Staubli VAL3: ros_server.pjx

--- ros_server.pjx ---
Parameters version=s7.7.2 stackSize=5000 millimeterUnit=true
Program file=atan2.pgx
Program file=dataReceiver.pgx
Program file=dataStreamer.pgx
Program file=decodeMsgBody.pgx
Program file=decodeMsgHeader.pgx
Program file=decTrajPtCartesian.pgx
Program file=decTrajPtJoint.pgx
Program file=decTrajPtJointFull.pgx
Program file=encodeAck.pgx
Program file=encodeJState.pgx
Program file=encodeStatus.pgx
Program file=encPrefixHeader.pgx
Program file=encTrajPtCartesianAck.pgx
Program file=encTrajPtJointAck.pgx
Program file=encTrajPtJointFAck.pgx
Program file=fetchStatus.pgx
Program file=initParams.pgx
Program file=motionControl.pgx
Program file=pushMotion.pgx
Program file=recvData.pgx
Program file=recvHeartbeat.pgx
Program file=recvMsgBody.pgx
Program file=recvMsgHeader.pgx
Program file=recvTrajPtCartesian.pgx
Program file=recvTrajPtJoint.pgx
Program file=recvTrajPtJointFull.pgx
Program file=screenUpdate.pgx
Program file=sendAck.pgx
Program file=sendData.pgx
Program file=sendRosMsg.pgx
Program file=setupRosMsgs.pgx
Program file=start.pgx
Program file=stop.pgx
Program file=toJointArrayRad.pgx
Program file=toJointRxDeg.pgx
Program file=toPointRxEuler.pgx
Program file=toPointRxMillis.pgx
Data file=ros_server.dtx
Library alias=libQueueFuncs path=Disk://ros_libs/QueueFuncs/QueueFuncs.pjx
Type name=RosSimpleMsg path=Disk://ros_libs/RosSimpleMsg/RosSimpleMsg.pjx
Type name=RobotStatusMsg path=Disk://ros_libs/RobotStatusMsg/RobotStatusMsg.pjx
Type name=CartesianTrajPtMsg path=Disk://ros_libs/CartesianTrajPtMsg/CartesianTrajPtMsg.pjx
Type name=JointStateMsg path=Disk://ros_libs/JointStateMsg/JointStateMsg.pjx
Type name=JointTrajPtMsg path=Disk://ros_libs/JointTrajPtMsg/JointTrajPtMsg.pjx
Type name=JointTrajPtFMsg path=Disk://ros_libs/JointTrajPtFMsg/JointTrajPtFMsg.pjx
Type name=JointFbkMsg path=Disk://ros_libs/JointFbkMsg/JointFbkMsg.pjx
Type name=MotionCmd path=Disk://ros_libs/MotionCmd/MotionCmd.pjx
Type name=Header path=Disk://ros_libs/Header/Header.pjx
Type name=Prefix path=Disk://ros_libs/Prefix/Prefix.pjx
Type name=Body path=Disk://ros_libs/Body/Body.pjx
Type name=Queue path=Disk://ros_libs/Queue/Queue.pjx

--- ros_server.dtx ---
public bool bFbkOverrun
public bool bMotionOverrun
public sio siTcpIpFbk = {link=Socket\Feedback}
public sio siTcpIpMotion = {link=Socket\Motion}
public string sStreamTaskName = "publisher"
public string sMotionTaskName
public RosSimpleMsg rosGenericMsg
  [0]
    Header header
      [0]
        num nMsgType
        num nCommType
        num nReplyCode
        num nData[12]
    Prefix prefix
      [0]
        num nLength
        num nData[4]
public tool tTool = {fatherId=flange[0], ioLink=valve1}
public string sTrajPtTaskName
public bool bTrajPtOverrun
public RobotStatusMsg rosStatusMsg
  [0]
    Body body
      [0]
        num nData[28]
    Header header
      [0]
        num nMsgType
        num nCommType
        num nReplyCode
        num nData[12]
    Prefix prefix
      [0]
        num nLength
        num nData[4]
    RobotStatus robotStatus
      [0]
        num nDrivesPowered
        num nEStopped
        num nErrorCode
        num nInError
        num nInMotion
        num nMode
        num nMotionPossible
public JointStateMsg rosJointMsg
  [0]
    Header header
      [0]
        num nMsgType
        num nCommType
        num nReplyCode
        num nData[12]
    Body body
      [0]
        num nData[44]
    JointState jointState
      [0]
        num nSeq
        num nJoints[10]
    Prefix prefix
      [0]
        num nLength
        num nData[4]
public JointTrajPtMsg rosTrajPtMsg
  [0]
    Header header
      [0]
        num nMsgType
        num nCommType
        num nReplyCode
        num nData[12]
    JointTrajPt jointTrajPt
      [0]
        num nSeq
        num nJoints[10]
        num nVelocity
        num nDuration
    Prefix prefix
      [0]
        num nLength
        num nData[4]
    Body body
      [0]
        num nData[52]
public JointTrajPtFMsg rosTrajPtFMsg
  [0]
    Header header
      [0]
        num nMsgType
        num nCommType
        num nReplyCode
        num nData[12]
    Prefix prefix
      [0]
        num nLength
        num nData[4]
    JointTrajPtFull jointTrajPtFull
      [0]
        num nRobotId
        num nSeq
        num nValidFields
        num nTime
        num nPositions[10]
        num nVelocities[10]
        num nAccelerations[10]
    Body body
      [0]
        num nData[136]
public JointFbkMsg rosJointFbkMsg
  [0]
    Header header
      [0]
        num nMsgType
        num nCommType
        num nReplyCode
        num nData[12]
    Prefix prefix
      [0]
        num nLength
        num nData[4]
    JointFeedback jointFeedback
      [0]
        num nRobotId
        num nValidFields
        num nTime
        num nPositions[10]
        num nVelocities[10]
        num nAccelerations[10]
    Body body
      [0]
        num nData[132]
public JointTrajPtFMsg rosTrajPtFAck
  [0]
    Header header
      [0]
        num nMsgType
        num nCommType
        num nReplyCode
        num nData[12]
    Prefix prefix
      [0]
        num nLength
        num nData[4]
    JointTrajPtFull jointTrajPtFull
      [0]
        num nRobotId
        num nSeq
        num nValidFields
        num nTime
        num nPositions[10]
        num nVelocities[10]
        num nAccelerations[10]
    Body body
      [0]
        num nData[136]
public JointTrajPtMsg rosTrajPtAck
  [0]
    Header header
      [0]
        num nMsgType
        num nCommType
        num nReplyCode
        num nData[12]
    JointTrajPt jointTrajPt
      [0]
        num nSeq
        num nJoints[10]
        num nVelocity
        num nDuration
    Prefix prefix
      [0]
        num nLength
        num nData[4]
    Body body
      [0]
        num nData[52]
public bool bScreenOverrun
public string sScreenTaskName
public num nInConnFlag
public num nOutConnFlag
public screen scDebug
public screen scMonitor
public string sHtbtTaskName
public num nPtsPopped
public bool bStopNow
public num nMotionProgress
public num nMoveId
public num nMovePts
public num nElapsedTime
public num nHeaderTime
public bool bOverwriteVel
public Queue qMoveBuffer
  [0]
    num nPush
    num nPop
    num nElems
    MotionCmd buffer[10]
      [0]
        mdesc mDesc = {leave=0, reach=0}
        num nDuration
        num nSequence
        num nMoveType
        jointRx jJointRx
        pointRx pPointRx
      [1]
        mdesc mDesc = {leave=0, reach=0}
        num nDuration
        num nSequence
        num nMoveType
        jointRx jJointRx
        pointRx pPointRx
      [2]
        mdesc mDesc = {leave=0, reach=0}
        num nDuration
        num nSequence
        num nMoveType
        jointRx jJointRx
        pointRx pPointRx
      [3]
        mdesc mDesc = {leave=0, reach=0}
        num nDuration
        num nSequence
        num nMoveType
        jointRx jJointRx
        pointRx pPointRx
      [4]
        mdesc mDesc = {leave=0, reach=0}
        num nDuration
        num nSequence
        num nMoveType
        jointRx jJointRx
        pointRx pPointRx
      [5]
        mdesc mDesc = {leave=0, reach=0}
        num nDuration
        num nSequence
        num nMoveType
        jointRx jJointRx
        pointRx pPointRx
      [6]
        mdesc mDesc = {leave=0, reach=0}
        num nDuration
        num nSequence
        num nMoveType
        jointRx jJointRx
        pointRx pPointRx
      [7]
        mdesc mDesc = {leave=0, reach=0}
        num nDuration
        num nSequence
        num nMoveType
        jointRx jJointRx
        pointRx pPointRx
      [8]
        mdesc mDesc = {leave=0, reach=0}
        num nDuration
        num nSequence
        num nMoveType
        jointRx jJointRx
        pointRx pPointRx
      [9]
        mdesc mDesc = {leave=0, reach=0}
        num nDuration
        num nSequence
        num nMoveType
        jointRx jJointRx
        pointRx pPointRx
public Queue qTrajPtBuffer
  [0]
    num nPush
    num nPop
    num nElems
    MotionCmd buffer[10]
      [0]
        mdesc mDesc = {leave=0, reach=0}
        num nDuration
        num nSequence
        num nMoveType
        jointRx jJointRx
        pointRx pPointRx
      [1]
        mdesc mDesc = {leave=0, reach=0}
        num nDuration
        num nSequence
        num nMoveType
        jointRx jJointRx
        pointRx pPointRx
      [2]
        mdesc mDesc = {leave=0, reach=0}
        num nDuration
        num nSequence
        num nMoveType
        jointRx jJointRx
        pointRx pPointRx
      [3]
        mdesc mDesc = {leave=0, reach=0}
        num nDuration
        num nSequence
        num nMoveType
        jointRx jJointRx
        pointRx pPointRx
      [4]
        mdesc mDesc = {leave=0, reach=0}
        num nDuration
        num nSequence
        num nMoveType
        jointRx jJointRx
        pointRx pPointRx
      [5]
        mdesc mDesc = {leave=0, reach=0}
        num nDuration
        num nSequence
        num nMoveType
        jointRx jJointRx
        pointRx pPointRx
      [6]
        mdesc mDesc = {leave=0, reach=0}
        num nDuration
        num nSequence
        num nMoveType
        jointRx jJointRx
        pointRx pPointRx
      [7]
        mdesc mDesc = {leave=0, reach=0}
        num nDuration
        num nSequence
        num nMoveType
        jointRx jJointRx
        pointRx pPointRx
      [8]
        mdesc mDesc = {leave=0, reach=0}
        num nDuration
        num nSequence
        num nMoveType
        jointRx jJointRx
        pointRx pPointRx
      [9]
        mdesc mDesc = {leave=0, reach=0}
        num nDuration
        num nSequence
        num nMoveType
        jointRx jJointRx
        pointRx pPointRx
public CartesianTrajPtMsg rosTrajPtCartesianMsg
  [0]
    Header header
      [0]
        num nMsgType
        num nCommType
        num nReplyCode
        num nData[12]
    CartesianTrajPt cartesianTrajPt
      [0]
        num nSeq
        num nPosition[3]
        num nOrientation[4]
        num nVelocity
        num nAcceleration
        num nBlendingRadius
        num nDuration
    Prefix prefix
      [0]
        num nLength
        num nData[4]
    Body body
      [0]
        num nData[48]
public CartesianTrajPtMsg rosTrajPtCartesianAck
  [0]
    Header header
      [0]
        num nMsgType
        num nCommType
        num nReplyCode
        num nData[12]
    CartesianTrajPt cartesianTrajPt
      [0]
        num nSeq
        num nPosition[3]
        num nOrientation[4]
        num nVelocity
        num nAcceleration
        num nBlendingRadius
        num nDuration
    Prefix prefix
      [0]
        num nLength
        num nData[4]
    Body body
      [0]
        num nData[48]
public pointRx pMovePointRx = {x=1, y=1, z=1, fatherId=world[0]}
public num nDeg2Rad = 0.01745329251
public num nRad2Deg = 57.2957795131

--- start.pgx ---
program start()
  local num l_nFbkPeriod
  local num l_nMotionPeriod
  local num l_nTrajPeriod
  local num l_nScreenUpdate
begin
  // Copyright (c) 2016, Ocado Technology - Robotics Research Team
  //
  // Licensed under the Apache License, Version 2.0 (the "License");
  // you may not use this file except in compliance with the License.
  // You may obtain a copy of the License at
  //
  //     http://www.apache.org/licenses/LICENSE-2.0
  //
  // Unless required by applicable law or agreed to in writing, software
  // distributed under the License is distributed on an "AS IS" BASIS,
  // WITHOUT WARRANTIES OR CONDITIONS OF ANY KIND, either express or implied.
  // See the License for the specific language governing permissions and
  // limitations under the License.



  // feedback task will run every 20ms (50Hz)
  l_nFbkPeriod=0.02
  //l_nFbkPeriod = 0.032 // 30Hz
  //l_nFbkPeriod = 0.05  // 20Hz
  //l_nFbkPeriod = 1.0   //  1Hz

  // motion control task will run every 4ms (250Hz)
  l_nMotionPeriod = 0.004
  //l_nMotionPeriod=0.012  // 83Hz
  //l_nMotionPeriod = 0.05 // 20Hz

  // data (trajectory) reception task will run every 4ms (250Hz)
  l_nTrajPeriod = 0.004
  // not in use at the moment
  l_nScreenUpdate = 1.0

  sStreamTaskName = "streamerTask"
  sTrajPtTaskName = "trajPtTask"
  sMotionTaskName = "motionTask"
  sScreenTaskName = "screenTask"
  sHtbtTaskName = "htbtTask"

  // initialise TCP/IP parameters
  call initParams()
  // setup prefix and header of ROS messages
  call setupRosMsgs()

  // socket connection status flags: initially disconnected
  nInConnFlag = 0
  nOutConnFlag = 0

  // flag defining whether velocity to be overwritten to max. vel.
  bOverwriteVel = false

  nPtsPopped = 0
  nMovePts = 0

  // flush buffer of incoming socket
  clearBuffer(siTcpIpMotion)
  // flush buffer of outgoing socket
  clearBuffer(siTcpIpFbk)

  // check if robot is not in emergency stop and wait until estop is reset
  if (esStatus() == 2)
    popUpMsg("Please reset E-Stop")
    wait(esStatus() < 2)
  endIf

  // before anything else, enable power (only works if robot is in remote mode)
  if (!isPowered())
    if (workingMode() >= 4)
      do
        enablePower()
        delay(2)
      until isPowered()
    else
      popUpMsg("Power must be enabled manually")
    endIf
  endIf

  // reset motion, potentially setting a start joint position for calling autoConnect() in the future
  resetMotion()

  // create joint state and robot status streamer task to send data to industrial_robot_client
  taskCreateSync sStreamTaskName, l_nFbkPeriod, bFbkOverrun, dataStreamer()

  // create trajectory point task to receive data from industrial_robot_client
  taskCreateSync sTrajPtTaskName, l_nTrajPeriod, bTrajPtOverrun, dataReceiver()
  //taskCreate sTrajPtTaskName, 100, dataReceiver()

  // create motion task to synchronously apply motion commands to robot
  taskCreateSync sMotionTaskName, l_nMotionPeriod, bMotionOverrun, motionControl()

  // create synchronous task to update screen
  //taskCreateSync sScreenTaskName, l_nScreenUpdate, bScreenOverrun, screenUpdate()
  taskCreate sScreenTaskName, 10, screenUpdate()

  // create asynchronous task to receive heartbeat on port 11002
  taskCreate sHtbtTaskName, 10, recvHeartbeat()

  logMsg("ROS-I Server started")

end

--- atan2.pgx ---
public program atan2(num x_nY, num x_nX, num& x_nResult)
begin
  if x_nX > 0
      x_nResult = atan(x_nY / x_nX)
  elseIf (x_nX < 0) and (x_nY >= 0)
      x_nResult = atan(x_nY / x_nX) + 180.0
  elseIf (x_nX < 0) and (x_nY < 0)
      x_nResult = atan(x_nY / x_nX) - 180.0
  elseIf (x_nX==0) and (x_nY > 0)
      x_nResult = 90.0
  elseIf (x_nX==0) and (x_nY < 0)
      x_nResult = -90.0
  elseIf (x_nX==0) and (x_nY==0)
      x_nResult = 0
  endIf
end

--- decodeMsgBody.pgx ---
public program decodeMsgBody(num& x_nMsgRecvState)
  local bool l_bFlag
begin
  // Copyright (c) 2016, Ocado Technology - Robotics Research Team
  //
  // Licensed under the Apache License, Version 2.0 (the "License");
  // you may not use this file except in compliance with the License.
  // You may obtain a copy of the License at
  //
  //     http://www.apache.org/licenses/LICENSE-2.0
  //
  // Unless required by applicable law or agreed to in writing, software
  // distributed under the License is distributed on an "AS IS" BASIS,
  // WITHOUT WARRANTIES OR CONDITIONS OF ANY KIND, either express or implied.
  // See the License for the specific language governing permissions and
  // limitations under the License.



  l_bFlag=false

  switch rosGenericMsg.header.nMsgType
    case 11
      call decTrajPtJoint(l_bFlag)
    break
    case 14
      call decTrajPtJointFull(l_bFlag)
    break
    case 31
      call decTrajPtCartesian(l_bFlag)
    break
    default
    break
  endSwitch

  if (l_bFlag == true)
    // move on to state 4: push motion into buffer
    x_nMsgRecvState=4
  else
    // error whilst decoding msg body...
    if (rosGenericMsg.header.nCommType==2)
      switch rosGenericMsg.header.nMsgType
        case 11
          rosTrajPtAck.header.nReplyCode=2
        break
        case 14
          rosTrajPtFAck.header.nReplyCode=2
        break
        case 31
          rosTrajPtCartesianAck.header.nReplyCode=2
        break
        default
        break
      endSwitch
      // jump to state 5: sendAck()
      x_nMsgRecvState=5
    else
      // reset state machine, since no ACK is required
      x_nMsgRecvState=0
    endIf
  endIf
end

--- decTrajPtCartesian.pgx ---
public program decTrajPtCartesian(bool& x_bFlag)
  local num l_nIndex
  local num l_nRetVal
begin
  // decode message ID 31 body (data)

  // assume failure to decode
  rosTrajPtCartesianAck.header.nReplyCode=2

  // sequence
  l_nRetVal=fromBinary(rosTrajPtCartesianMsg.body.nData,4,"-4l",rosTrajPtCartesianMsg.cartesianTrajPt.nSeq)
  if(l_nRetVal!=1)
    x_bFlag=false
    return
  endIf

  // position[3]
  for l_nIndex=0 to 2 step 1
    l_nRetVal=fromBinary(rosTrajPtCartesianMsg.body.nData[(l_nIndex*4)+4],4,"4.0l",rosTrajPtCartesianMsg.cartesianTrajPt.nPosition[l_nIndex])
    if(l_nRetVal!=1)
      x_bFlag=false
      return
    endIf
  endFor

  // orientation[4]
  for l_nIndex=0 to 3 step 1
    l_nRetVal=fromBinary(rosTrajPtCartesianMsg.body.nData[(l_nIndex*4)+16],4,"4.0l",rosTrajPtCartesianMsg.cartesianTrajPt.nOrientation[l_nIndex])
    if(l_nRetVal!=1)
      x_bFlag=false
      return
    endIf
  endFor

  // velocity
  l_nRetVal=fromBinary(rosTrajPtCartesianMsg.body.nData[32],4,"4.0l",rosTrajPtCartesianMsg.cartesianTrajPt.nVelocity)
  if(l_nRetVal!=1)
    x_bFlag=false
    return
  endIf

  // acceleration
  l_nRetVal=fromBinary(rosTrajPtCartesianMsg.body.nData[36],4,"4.0l",rosTrajPtCartesianMsg.cartesianTrajPt.nAcceleration)
  if(l_nRetVal!=1)
    x_bFlag=false
    return
  endIf

  // blending radius
  l_nRetVal=fromBinary(rosTrajPtCartesianMsg.body.nData[40],4,"4.0l",rosTrajPtCartesianMsg.cartesianTrajPt.nBlendingRadius)
  if(l_nRetVal!=1)
    x_bFlag=false
    return
  endIf

  // duration
  l_nRetVal=fromBinary(rosTrajPtCartesianMsg.body.nData[44],4,"4.0l",rosTrajPtCartesianMsg.cartesianTrajPt.nDuration)
  if(l_nRetVal!=1)
    x_bFlag=false
    return
  endIf

  // decoding successful
  rosTrajPtCartesianAck.header.nReplyCode=1
  rosTrajPtCartesianAck.cartesianTrajPt.nSeq=rosTrajPtCartesianMsg.cartesianTrajPt.nSeq
  x_bFlag=true
end

--- decTrajPtJoint.pgx ---
public program decTrajPtJoint(bool& x_bFlag)
  local num l_nIndex
  local num l_nRetVal
begin
  // Copyright (c) 2016, Ocado Technology - Robotics Research Team
  //
  // Licensed under the Apache License, Version 2.0 (the "License");
  // you may not use this file except in compliance with the License.
  // You may obtain a copy of the License at
  //
  //     http://www.apache.org/licenses/LICENSE-2.0
  //
  // Unless required by applicable law or agreed to in writing, software
  // distributed under the License is distributed on an "AS IS" BASIS,
  // WITHOUT WARRANTIES OR CONDITIONS OF ANY KIND, either express or implied.
  // See the License for the specific language governing permissions and
  // limitations under the License.



  // decode message ID 11 body (data)

  // assume failure to decode
  rosTrajPtAck.header.nReplyCode=2

  // sequence
  l_nRetVal=fromBinary(rosTrajPtMsg.body.nData,4,"-4l",rosTrajPtMsg.jointTrajPt.nSeq)
  if (l_nRetVal!=1)
    x_bFlag=false
    return
  endIf

  // joints[10]
  for l_nIndex=0 to 9 step 1
    l_nRetVal=fromBinary(rosTrajPtMsg.body.nData[(l_nIndex*4)+4],4,"4.0l",rosTrajPtMsg.jointTrajPt.nJoints[l_nIndex])
    if (l_nRetVal!=1)
      x_bFlag=false
      return
    endIf
  endFor

  // velocity
  l_nRetVal=fromBinary(rosTrajPtMsg.body.nData[44],4,"4.0l",rosTrajPtMsg.jointTrajPt.nVelocity)
  if (l_nRetVal!=1)
    x_bFlag=false
    return
  endIf

  // duration
  l_nRetVal=fromBinary(rosTrajPtMsg.body.nData[48],4,"4.0l",rosTrajPtMsg.jointTrajPt.nDuration)
  if (l_nRetVal!=1)
    x_bFlag=false
    return
  endIf

  // decoding successful
  rosTrajPtAck.header.nReplyCode=1
  rosTrajPtAck.jointTrajPt.nSeq=rosTrajPtMsg.jointTrajPt.nSeq
  x_bFlag=true
end

--- decTrajPtJointFull.pgx ---
public program decTrajPtJointFull(bool& x_bFlag)
  local num l_nIndex
  local num l_nRetVal
begin
  // Copyright (c) 2016, Ocado Technology - Robotics Research Team
  //
  // Licensed under the Apache License, Version 2.0 (the "License");
  // you may not use this file except in compliance with the License.
  // You may obtain a copy of the License at
  //
  //     http://www.apache.org/licenses/LICENSE-2.0
  //
  // Unless required by applicable law or agreed to in writing, software
  // distributed under the License is distributed on an "AS IS" BASIS,
  // WITHOUT WARRANTIES OR CONDITIONS OF ANY KIND, either express or implied.
  // See the License for the specific language governing permissions and
  // limitations under the License.



  // decode message ID 14 body (data)

  // assume failure to decode
  rosTrajPtFAck.header.nReplyCode=2

  // robotId
  l_nRetVal=fromBinary(rosTrajPtFMsg.body.nData,4,"-4l",rosTrajPtFMsg.jointTrajPtFull.nRobotId)
  if (l_nRetVal!=1)
    x_bFlag=false
    return
  endIf

  // sequence
  l_nRetVal=fromBinary(rosTrajPtFMsg.body.nData,4,"-4l",rosTrajPtFMsg.jointTrajPtFull.nSeq)
  if (l_nRetVal!=1)
    x_bFlag=false
    return
  endIf

  // valid fields
  l_nRetVal=fromBinary(rosTrajPtFMsg.body.nData,4,"-4l",rosTrajPtFMsg.jointTrajPtFull.nValidFields)
  if (l_nRetVal!=1)
    x_bFlag=false
    return
  endIf

  // time
  l_nRetVal=fromBinary(rosTrajPtFMsg.body.nData,4,"4.0l",rosTrajPtFMsg.jointTrajPtFull.nTime)
  if (l_nRetVal!=1)
    x_bFlag=false
    return
  endIf

  // positions[10]
  for l_nIndex=0 to 9 step 1
    l_nRetVal=fromBinary(rosTrajPtFMsg.body.nData[(l_nIndex*4)+16],4,"4.0l",rosTrajPtFMsg.jointTrajPtFull.nPositions[l_nIndex])
    if (l_nRetVal!=1)
      x_bFlag=false
      return
    endIf
  endFor

  // velocities[10]
  for l_nIndex=0 to 9 step 1
    l_nRetVal=fromBinary(rosTrajPtFMsg.body.nData[(l_nIndex*4)+56],4,"4.0l",rosTrajPtFMsg.jointTrajPtFull.nVelocities[l_nIndex])
    if (l_nRetVal!=1)
      x_bFlag=false
      return
    endIf
  endFor

  // accelerations[10]
  for l_nIndex=0 to 9 step 1
    l_nRetVal=fromBinary(rosTrajPtFMsg.body.nData[(l_nIndex*4)+96],4,"4.0l",rosTrajPtFMsg.jointTrajPtFull.nAccelerations[l_nIndex])
    if (l_nRetVal!=1)
      x_bFlag=false
      return
    endIf
  endFor

  // decoding successful
  rosTrajPtFAck.header.nReplyCode=1
  rosTrajPtFAck.jointTrajPtFull.nSeq=rosTrajPtFMsg.jointTrajPtFull.nSeq
  x_bFlag=true
end

--- encodeAck.pgx ---
public program encodeAck()
begin
  // Copyright (c) 2016, Ocado Technology - Robotics Research Team
  //
  // Licensed under the Apache License, Version 2.0 (the "License");
  // you may not use this file except in compliance with the License.
  // You may obtain a copy of the License at
  //
  //     http://www.apache.org/licenses/LICENSE-2.0
  //
  // Unless required by applicable law or agreed to in writing, software
  // distributed under the License is distributed on an "AS IS" BASIS,
  // WITHOUT WARRANTIES OR CONDITIONS OF ANY KIND, either express or implied.
  // See the License for the specific language governing permissions and
  // limitations under the License.



  switch rosGenericMsg.header.nMsgType
    case 11
      call encTrajPtJointAck()
    break
    case 14
      call encTrajPtJointFAck()
    break
    case 31
      call encTrajPtCartesianAck()
    break
    default
    break
  endSwitch
end

--- encTrajPtCartesianAck.pgx ---
public program encTrajPtCartesianAck()
begin
  // encode 'prefix' and 'header'
  call encPrefixHeader(rosTrajPtCartesianAck.prefix, rosTrajPtCartesianAck.header)

  // encode 'sequence' variable of body message (data)
  toBinary(rosTrajPtCartesianAck.cartesianTrajPt.nSeq,1,"-4l",rosTrajPtCartesianAck.body.nData)

  // encodings of all other fields ignored to save CPU time, since values are all zeros
end

--- encTrajPtJointAck.pgx ---
public program encTrajPtJointAck()
begin
  // Copyright (c) 2016, Ocado Technology - Robotics Research Team
  //
  // Licensed under the Apache License, Version 2.0 (the "License");
  // you may not use this file except in compliance with the License.
  // You may obtain a copy of the License at
  //
  //     http://www.apache.org/licenses/LICENSE-2.0
  //
  // Unless required by applicable law or agreed to in writing, software
  // distributed under the License is distributed on an "AS IS" BASIS,
  // WITHOUT WARRANTIES OR CONDITIONS OF ANY KIND, either express or implied.
  // See the License for the specific language governing permissions and
  // limitations under the License.



  // encode 'prefix' and 'header'
  call encPrefixHeader(rosTrajPtAck.prefix, rosTrajPtAck.header)

  // encode 'sequence' variable of body message (data)
  toBinary(rosTrajPtAck.jointTrajPt.nSeq,1,"-4l",rosTrajPtAck.body.nData)

  // encodings of 'joints[10]', 'velocity' and 'duration' ignored to save CPU time, since values are all zeros
end

--- encTrajPtJointFAck.pgx ---
public program encTrajPtJointFAck()
begin
  // Copyright (c) 2016, Ocado Technology - Robotics Research Team
  //
  // Licensed under the Apache License, Version 2.0 (the "License");
  // you may not use this file except in compliance with the License.
  // You may obtain a copy of the License at
  //
  //     http://www.apache.org/licenses/LICENSE-2.0
  //
  // Unless required by applicable law or agreed to in writing, software
  // distributed under the License is distributed on an "AS IS" BASIS,
  // WITHOUT WARRANTIES OR CONDITIONS OF ANY KIND, either express or implied.
  // See the License for the specific language governing permissions and
  // limitations under the License.



  // encode 'prefix' and 'header'
  call encPrefixHeader(rosTrajPtFAck.prefix, rosTrajPtFAck.header)

  // encode body message (data)
  toBinary(rosTrajPtFAck.jointTrajPtFull.nRobotId,1,"-4l",rosTrajPtFAck.body.nData)
  toBinary(rosTrajPtFAck.jointTrajPtFull.nSeq,1,"-4l",rosTrajPtFAck.body.nData[4])

  // encodings of 'positions[10]', velocities[10]' and accelerations[10]' ignored to save CPU time, since values are all zeros
end

--- motionControl.pgx ---
public program motionControl()
  local MotionCmd l_mTrajPt
  local bool l_bFlag
  local MotionCmd l_motion
  local num l_nTime
  local bool l_bStopAndClean
  local num l_nElems
begin
  // Copyright (c) 2016, Ocado Technology - Robotics Research Team
  //
  // Licensed under the Apache License, Version 2.0 (the "License");
  // you may not use this file except in compliance with the License.
  // You may obtain a copy of the License at
  //
  //     http://www.apache.org/licenses/LICENSE-2.0
  //
  // Unless required by applicable law or agreed to in writing, software
  // distributed under the License is distributed on an "AS IS" BASIS,
  // WITHOUT WARRANTIES OR CONDITIONS OF ANY KIND, either express or implied.
  // See the License for the specific language governing permissions and
  // limitations under the License.



  nMoveId = -1

  while (true)
    // check connection status, and whether to stop motion
    if (nInConnFlag == 1 and nOutConnFlag == 1 and bStopNow == false)

      // process trajectory point from trajectory buffer
      call libQueueFuncs:getNumElems(qTrajPtBuffer, l_nElems)
      if (l_nElems > 0)
        call libQueueFuncs:pop(qTrajPtBuffer,l_mTrajPt, l_bFlag)
        if (l_bFlag == true)
          nPtsPopped = nPtsPopped + 1
          call libQueueFuncs:push(qMoveBuffer,l_mTrajPt,l_bFlag)
        endIf
      endIf

      // process motion command from move buffer
      // @TODO move buffer should have elements previously interpolated to ensure they are 4 ms apart
      call libQueueFuncs:getNumElems(qMoveBuffer, l_nElems)
      if (l_nElems > 0)
        call libQueueFuncs:pop(qMoveBuffer,l_motion,l_bFlag)
        if (l_bFlag == true)
          nMovePts = nMovePts + 1

          if l_motion.nMoveType >= 20 and l_motion.nMoveType < 30
            pMovePointRx.trsf = l_motion.pPointRx.trsf
          endIf

          // @TODO potentially set move id according to sequence value
          if l_motion.nMoveType == 10
            nMoveId = movej(l_motion.jJointRx, tTool, l_motion.mDesc)
          elseIf l_motion.nMoveType == 20
            nMoveId = movej(pMovePointRx, tTool, l_motion.mDesc)
          elseIf l_motion.nMoveType == 21
            nMoveId = movel(pMovePointRx, tTool, l_motion.mDesc)
          endIf
        endIf
      endIf
    else
      // stop immediately -- resetMotion() also resets moveId
      resetMotion()
      // clear buffers
      call libQueueFuncs:clear(qTrajPtBuffer)
      call libQueueFuncs:clear(qMoveBuffer)
      bStopNow = false

      // debug
      nPtsPopped = 0
      nMovePts = 0
    endIf

    nMotionProgress = getMoveId()

    // sequence task
    delay(0)
  endWhile
end

--- pushMotion.pgx ---
public program pushMotion(num& x_nMsgRecvState)
  local bool l_bOk
  local bool l_bWillMove
  local num l_nCounter
  local num l_nJointError
  local MotionCmd l_mTrajPt
begin
  // Copyright (c) 2016, Ocado Technology - Robotics Research Team
  //
  // Licensed under the Apache License, Version 2.0 (the "License");
  // you may not use this file except in compliance with the License.
  // You may obtain a copy of the License at
  //
  //     http://www.apache.org/licenses/LICENSE-2.0
  //
  // Unless required by applicable law or agreed to in writing, software
  // distributed under the License is distributed on an "AS IS" BASIS,
  // WITHOUT WARRANTIES OR CONDITIONS OF ANY KIND, either express or implied.
  // See the License for the specific language governing permissions and
  // limitations under the License.

  // MoveType = 10: movej(jointRx)
  // MoveType = 20: movej(pointRx)
  // MoveType = 21: movel(pointRx)

  switch rosGenericMsg.header.nMsgType
    case 11
      l_mTrajPt.nMoveType = 10
      l_mTrajPt.nSequence=rosTrajPtMsg.jointTrajPt.nSeq

      // ROS joint position values are in rad, but VAL3 uses degrees
      call toJointRxDeg(rosTrajPtMsg.jointTrajPt.nJoints, l_mTrajPt.jJointRx)

      // from industrial_robot_client/src/joint_trajectory_interface.cpp
      // JointTrajectoryInterface::trajectory_to_msgs()
      // JointTrajectoryInterface::calc_speed()
      // velocity is converted to a scalar value representing % of max velocity,
      // such that 0.2 = 20% of maximum joint speed
      l_mTrajPt.mDesc.vel= limit((rosTrajPtMsg.jointTrajPt.nVelocity * 100), 0, 100)
      l_mTrajPt.nDuration=rosTrajPtMsg.jointTrajPt.nDuration

    break
    case 14
      l_mTrajPt.nMoveType = 10
      l_mTrajPt.nSequence=rosTrajPtFMsg.jointTrajPtFull.nSeq
      l_mTrajPt.nDuration=rosTrajPtFMsg.jointTrajPtFull.nTime

      // ROS joint position values are in rad, but VAL3 uses degrees
      call toJointRxDeg(rosTrajPtFMsg.jointTrajPtFull.nPositions, l_mTrajPt.jJointRx)

      // from industrial_robot_client/src/joint_trajectory_interface.cpp
      // JointTrajectoryInterface::trajectory_to_msgs()
      // JointTrajectoryInterface::calc_speed()
      // velocity is converted to a scalar value representing % of max velocity,
      // such that 0.2 = 20% of maximum joint speed
      l_mTrajPt.mDesc.vel= limit((rosTrajPtFMsg.jointTrajPtFull.nVelocities[0] * 100), 0, 100)
      // not sure about accelerations as yet
      l_mTrajPt.mDesc.accel=rosTrajPtFMsg.jointTrajPtFull.nAccelerations[0]
      l_mTrajPt.mDesc.decel=l_mTrajPt.mDesc.accel
    break
    case 31
      l_mTrajPt.nMoveType = 21
      l_mTrajPt.nSequence=rosTrajPtCartesianMsg.cartesianTrajPt.nSeq

      // ROS position is in meters but VAL3 uses millimeters
      call toPointRxMillis(rosTrajPtCartesianMsg.cartesianTrajPt.nPosition, l_mTrajPt.pPointRx)

      // ROS orientation is in quaternion (rad) but VAL3 uses euler angles
      call toPointRxEuler(rosTrajPtCartesianMsg.cartesianTrajPt.nOrientation, l_mTrajPt.pPointRx)

      // Read accel/decel values
      l_mTrajPt.mDesc.accel = limit(rosTrajPtCartesianMsg.cartesianTrajPt.nAcceleration, 0, 100)
      l_mTrajPt.mDesc.decel = l_mTrajPt.mDesc.accel

      // velocity is a scalar value representing % of max velocity,
      // such that 0.2 = 20% of maximum joint speed
      l_mTrajPt.mDesc.vel= limit((rosTrajPtCartesianMsg.cartesianTrajPt.nVelocity * 100), 0, 100)
      l_mTrajPt.nDuration=rosTrajPtMsg.jointTrajPt.nDuration

    break
    default
    break
  endSwitch

  // see github.com/ros-industrial/industrial_core/simple_message/include/simple_message/joint_traj_pt.h
  if (l_mTrajPt.nSequence==-4)
    // set flag to stop immediately
    bStopNow=true
  else
    // check whether velocity value should be overwritten with value set on teach pendant
    if (bOverwriteVel == true)
      // overwrite velocity (and acceleration - ?)
      l_mTrajPt.mDesc.vel = getMonitorSpeed()
      // explicitly setting accel and decel to VAL3 default values
      l_mTrajPt.mDesc.accel = 9999
      l_mTrajPt.mDesc.decel = 9999
    endIf
    // only push motion into buffer if not a STOP message
    // if it's a joint type of move
    //   and if joint positions are within software joint limits
    //   and if velocity is greater than zero (because movej() will not accept vel <= 0)
    // or if it's a point type of move
    //   and if velocity is greater than zero
    l_bWillMove = false
    if (l_mTrajPt.nMoveType >= 10 and l_mTrajPt.nMoveType < 20) and (isInRange(l_mTrajPt.jJointRx) and l_mTrajPt.mDesc.vel > 0)
      l_bWillMove = true
    elseIf (l_mTrajPt.nMoveType >= 20 and l_mTrajPt.nMoveType < 30) and l_mTrajPt.mDesc.vel > 0
      l_bWillMove = true
    endIf

    if (l_bWillMove == true)

      // Check if we need to power up before the first point of a sequence
      // This is only possible in remote mode.
      if (l_mTrajPt.nSequence == 0)
        // before move, check if we need to enable power
        // (only works if robot is in remote mode)
        if (workingMode() >= 4 and !isPowered())
            do
            enablePower()
            delay(1)
            until isPowered()
        endIf
      endIf

      call libQueueFuncs:push(qTrajPtBuffer,l_mTrajPt,l_bOk)
    else
      l_bOk = false
    endIf

    if (l_bOk==false)
      // could not push trajectory point into buffer
      // thus ACK should flag FAILURE, but only if comm type is request
      if (rosGenericMsg.header.nCommType==2)
        switch rosGenericMsg.header.nMsgType
          case 11
            rosTrajPtAck.header.nReplyCode=2
          break
          case 14
            rosTrajPtFAck.header.nReplyCode=2
          break
          case 31
            rosTrajPtCartesianAck.header.nReplyCode=2
          break
          default
          break
        endSwitch
      endIf
    endIf
  endIf
  // check whether ACK should be sent
  if (rosGenericMsg.header.nCommType == 2)
    // comm type request requires ACK
    x_nMsgRecvState = 5
  else
    // other comm types (e.g., topic) does not require ACK, hence skip state
    x_nMsgRecvState = 0
  endIf
end

--- recvMsgBody.pgx ---
public program recvMsgBody(num& x_nMsgRecvState)
  local bool l_bFlag
begin
  // Copyright (c) 2016, Ocado Technology - Robotics Research Team
  //
  // Licensed under the Apache License, Version 2.0 (the "License");
  // you may not use this file except in compliance with the License.
  // You may obtain a copy of the License at
  //
  //     http://www.apache.org/licenses/LICENSE-2.0
  //
  // Unless required by applicable law or agreed to in writing, software
  // distributed under the License is distributed on an "AS IS" BASIS,
  // WITHOUT WARRANTIES OR CONDITIONS OF ANY KIND, either express or implied.
  // See the License for the specific language governing permissions and
  // limitations under the License.



  l_bFlag=false

  switch rosGenericMsg.header.nMsgType
    case 11
      call recvTrajPtJoint(l_bFlag)
    break
    case 14
      call recvTrajPtJointFull(l_bFlag)
    break
    case 31
      call recvTrajPtCartesian(l_bFlag)
    break
    default
    break
  endSwitch

  if (l_bFlag == true)
    // move on to state 3: decode msg body
    x_nMsgRecvState=3
  else
    // error whilst receiving msg body, reset state machine
    x_nMsgRecvState=0
  endIf
end

--- recvTrajPtCartesian.pgx ---
public program recvTrajPtCartesian(bool& x_bFlag)
begin
  // attempt to receive message ID 31 data (prefix and header are in rosGenericMsg)
  rosTrajPtCartesianMsg.prefix.nLength=rosGenericMsg.prefix.nLength
  rosTrajPtCartesianMsg.header.nMsgType=rosGenericMsg.header.nMsgType
  rosTrajPtCartesianMsg.header.nCommType=rosGenericMsg.header.nCommType
  rosTrajPtCartesianMsg.header.nReplyCode=rosGenericMsg.header.nReplyCode

  call recvData(siTcpIpMotion,rosTrajPtCartesianMsg.body.nData,nInConnFlag,x_bFlag)
end

--- recvTrajPtJoint.pgx ---
public program recvTrajPtJoint(bool& x_bFlag)
begin
  // Copyright (c) 2016, Ocado Technology - Robotics Research Team
  //
  // Licensed under the Apache License, Version 2.0 (the "License");
  // you may not use this file except in compliance with the License.
  // You may obtain a copy of the License at
  //
  //     http://www.apache.org/licenses/LICENSE-2.0
  //
  // Unless required by applicable law or agreed to in writing, software
  // distributed under the License is distributed on an "AS IS" BASIS,
  // WITHOUT WARRANTIES OR CONDITIONS OF ANY KIND, either express or implied.
  // See the License for the specific language governing permissions and
  // limitations under the License.



  // attempt to receive message ID 11 data (prefix and header are in rosGenericMsg)
  rosTrajPtMsg.prefix.nLength=rosGenericMsg.prefix.nLength
  rosTrajPtMsg.header.nMsgType=rosGenericMsg.header.nMsgType
  rosTrajPtMsg.header.nCommType=rosGenericMsg.header.nCommType
  rosTrajPtMsg.header.nReplyCode=rosGenericMsg.header.nReplyCode

  call recvData(siTcpIpMotion,rosTrajPtMsg.body.nData,nInConnFlag,x_bFlag)
end

--- recvTrajPtJointFull.pgx ---
public program recvTrajPtJointFull(bool& x_bFlag)
begin
  // Copyright (c) 2016, Ocado Technology - Robotics Research Team
  //
  // Licensed under the Apache License, Version 2.0 (the "License");
  // you may not use this file except in compliance with the License.
  // You may obtain a copy of the License at
  //
  //     http://www.apache.org/licenses/LICENSE-2.0
  //
  // Unless required by applicable law or agreed to in writing, software
  // distributed under the License is distributed on an "AS IS" BASIS,
  // WITHOUT WARRANTIES OR CONDITIONS OF ANY KIND, either express or implied.
  // See the License for the specific language governing permissions and
  // limitations under the License.



  // receive message ID 14 data (prefix and header are in rosGenericMsg)
  rosTrajPtFMsg.prefix.nLength=rosGenericMsg.prefix.nLength
  rosTrajPtFMsg.header.nMsgType=rosGenericMsg.header.nMsgType
  rosTrajPtFMsg.header.nCommType=rosGenericMsg.header.nCommType
  rosTrajPtFMsg.header.nReplyCode=rosGenericMsg.header.nReplyCode

  call recvData(siTcpIpMotion,rosTrajPtFMsg.body.nData,nInConnFlag,x_bFlag)
end

--- sendAck.pgx ---
public program sendAck(num& x_nMsgRecvState)
begin
  // Copyright (c) 2016, Ocado Technology - Robotics Research Team
  //
  // Licensed under the Apache License, Version 2.0 (the "License");
  // you may not use this file except in compliance with the License.
  // You may obtain a copy of the License at
  //
  //     http://www.apache.org/licenses/LICENSE-2.0
  //
  // Unless required by applicable law or agreed to in writing, software
  // distributed under the License is distributed on an "AS IS" BASIS,
  // WITHOUT WARRANTIES OR CONDITIONS OF ANY KIND, either express or implied.
  // See the License for the specific language governing permissions and
  // limitations under the License.



  switch rosGenericMsg.header.nMsgType
    case 11
      call sendRosMsg(siTcpIpMotion, rosTrajPtAck.prefix, rosTrajPtAck.header, rosTrajPtAck.body, nInConnFlag)
    break
    case 14
      call sendRosMsg(siTcpIpMotion, rosTrajPtFAck.prefix, rosTrajPtFAck.header, rosTrajPtFAck.body, nInConnFlag)
    break
    case 31
      call sendRosMsg(siTcpIpMotion, rosTrajPtCartesianAck.prefix, rosTrajPtCartesianAck.header, rosTrajPtCartesianAck.body, nInConnFlag)
    break
    default
    break
  endSwitch

  // regardless of result from sending ACK
  // reset state machine to receive new messages
  x_nMsgRecvState=0
end

--- setupRosMsgs.pgx ---
public program setupRosMsgs()
begin
  // Copyright (c) 2016, Ocado Technology - Robotics Research Team
  //
  // Licensed under the Apache License, Version 2.0 (the "License");
  // you may not use this file except in compliance with the License.
  // You may obtain a copy of the License at
  //
  //     http://www.apache.org/licenses/LICENSE-2.0
  //
  // Unless required by applicable law or agreed to in writing, software
  // distributed under the License is distributed on an "AS IS" BASIS,
  // WITHOUT WARRANTIES OR CONDITIONS OF ANY KIND, either express or implied.
  // See the License for the specific language governing permissions and
  // limitations under the License.



  // Joint state message (ID 10)
  // prefix length = 12 + 44
  rosJointMsg.prefix.nLength=56
  rosJointMsg.header.nMsgType=10
  rosJointMsg.header.nCommType=1
  rosJointMsg.header.nReplyCode=0
  // sequence
  rosJointMsg.jointState.nSeq=0



  // Joint trajectory point message (ID 11)
  // prefix length = 12 + 52
  rosTrajPtAck.prefix.nLength=64
  rosTrajPtAck.header.nMsgType=11
  rosTrajPtAck.header.nCommType=3
  // reply: 1 = success, 2 = failure
  rosTrajPtAck.header.nReplyCode=1
  // joints are assumed to be initiliased to zero

  // the message bellow will be filled upon reception
  rosTrajPtMsg.prefix.nLength=64



  // Robot status message (ID 13)
  // prefix length = 12 + 28
  rosStatusMsg.prefix.nLength=40
  rosStatusMsg.header.nMsgType=13
  rosStatusMsg.header.nCommType=1
  rosStatusMsg.header.nReplyCode=0



  // Joint trajectory point full message (ID 14)
  // prefix length = 12 + 136
  rosTrajPtFAck.prefix.nLength=148
  rosTrajPtFAck.header.nMsgType=14
  rosTrajPtFAck.header.nCommType=3
  // reply: 1 = success, 2 = failure
  rosTrajPtFAck.header.nReplyCode=1
  // body (data) assumed to be initialised to zero

  // the message bellow will be filled upon reception
  rosTrajPtFMsg.prefix.nLength=148

  // Cartesian trajectory point message (ID 31)
  // prefix length = 12 + 48
  rosTrajPtCartesianAck.prefix.nLength=60
  rosTrajPtCartesianAck.header.nMsgType=31
  rosTrajPtCartesianAck.header.nCommType=3
  // reply: 1 = success, 2 = failure
  rosTrajPtCartesianAck.header.nReplyCode=1
  // position, orientation, velocities, etc are assumed to be initiliased to zero

  // the message bellow will be filled upon reception
  rosTrajPtCartesianMsg.prefix.nLength=60


  // Joint feedback message (ID 15)
  // prefix length = 12 + 132
  rosJointFbkMsg.prefix.nLength=144
  rosJointFbkMsg.header.nMsgType=15
  rosJointFbkMsg.header.nCommType=1
  rosJointFbkMsg.header.nReplyCode=0
end

--- toJointArrayRad.pgx ---
public program toJointArrayRad(jointRx& x_jJointRx, num& x_nJointArray[])
begin
  // Copyright (c) 2016, Ocado Technology - Robotics Research Team
  //
  // Licensed under the Apache License, Version 2.0 (the "License");
  // you may not use this file except in compliance with the License.
  // You may obtain a copy of the License at
  //
  //     http://www.apache.org/licenses/LICENSE-2.0
  //
  // Unless required by applicable law or agreed to in writing, software
  // distributed under the License is distributed on an "AS IS" BASIS,
  // WITHOUT WARRANTIES OR CONDITIONS OF ANY KIND, either express or implied.
  // See the License for the specific language governing permissions and
  // limitations under the License.

  // assuming the remaining elements (6-9) have zeros assigned by default
  x_nJointArray[0] = x_jJointRx.j1 * nDeg2Rad
  x_nJointArray[1] = x_jJointRx.j2 * nDeg2Rad
  x_nJointArray[2] = x_jJointRx.j3 * nDeg2Rad
  x_nJointArray[3] = x_jJointRx.j4 * nDeg2Rad
  x_nJointArray[4] = x_jJointRx.j5 * nDeg2Rad
  x_nJointArray[5] = x_jJointRx.j6 * nDeg2Rad
end

--- toPointRxEuler.pgx ---
public program toPointRxEuler(num& x_nQuaternion[], pointRx& x_pPointRx)
  local num l_nT0
  local num l_nT1
  local num l_nT2
  local num l_nT3
  local num l_nT4
  local num l_nAtan2Res
  local num _EPS
  local num si
  local num sj
  local num sk
  local num ci
  local num cj
  local num ck
  local num M02
  local num M12
  local num M22
  local num cy
  local num ax
  local num ay
  local num az
begin
  _EPS = 1e-16

  l_nT0 = 2 * (x_nQuaternion[3] * x_nQuaternion[0] + x_nQuaternion[1] * x_nQuaternion[2])
  l_nT1 = 1 - 2 * (x_nQuaternion[0] * x_nQuaternion[0] + x_nQuaternion[1] * x_nQuaternion[1])
  call atan2(l_nT0, l_nT1, l_nAtan2Res)
  si = sin(l_nAtan2Res)
  ci = cos(l_nAtan2Res)

  l_nT2 = 2 * (x_nQuaternion[3] * x_nQuaternion[1] - x_nQuaternion[2] * x_nQuaternion[0])
  sj = limit(l_nT2, -1, 1)
  cj = cos(asin(sj))

  l_nT3 = 2 * (x_nQuaternion[3] * x_nQuaternion[2] + x_nQuaternion[0] * x_nQuaternion[1])
  l_nT4 = 1 - 2 * (x_nQuaternion[1] * x_nQuaternion[1] + x_nQuaternion[2] * x_nQuaternion[2])
  call atan2(l_nT3, l_nT4, l_nAtan2Res)
  sk = sin(l_nAtan2Res)
  ck = cos(l_nAtan2Res)

  // extrinsic2intrinsic
  M02 = sj * ci * ck + si * sk
  M12 = sj * ci * sk - si * ck
  M22 = cj * ci

  cy = sqrt(M22 * M22 + M12 * M12)

  if cy > _EPS
    call atan2(M12, M22, ax)
    call atan2(-M02, cy, ay)
    call atan2(sj * (si * ck) - (ci * sk), cj * ck, az)
  else
    ax = 0.0
    call atan2(-M02, cy, ay)
    call atan2(-cj * sk, sj * si * sk + ci * ck, az)
  endIf

  x_pPointRx.trsf.rx = ax * -1
  x_pPointRx.trsf.ry = ay * -1
  x_pPointRx.trsf.rz = az * -1

end

--- toPointRxMillis.pgx ---
public program toPointRxMillis(num& x_nPositionArray[], pointRx& x_pPointRx)
  local num l_nScaleFactor
begin
  l_nScaleFactor = 1000.0
  x_pPointRx.trsf.x = x_nPositionArray[0] * l_nScaleFactor
  x_pPointRx.trsf.y = x_nPositionArray[1] * l_nScaleFactor
  x_pPointRx.trsf.z = x_nPositionArray[2] * l_nScaleFactor
end
